PROGRAM MAIN
VAR
	a: INT;
	b: INT;
	c: INT;
	enable: BOOL;
	
END_VAR

IF enable THEN
	a:= b;
ELSE
	a:= c;
	
END_IF

END_PROGRAM

(* stored: Version 1.1.0.1, ProductVersion 3.1.4024.12
   POU MAIN: Id {86359209-05ee-48c8-92db-5782fc05259f}, SpecialFunc None *)
